# EPICS autosave request: aravisApp/Db/aravisCamera_settings.req
file "ADGenICam_settings.req", P=$(P), R=$(R)
$(P)$(R)ARPacketResendEnable
$(P)$(R)ARConvertPixelFormat
$(P)$(R)ARLeftShift
$(P)$(R)ARPacketTimeout
$(P)$(R)ARFrameRetention
